_CFC_ (* Continuous Function Chart, elements in execution order *)
#0 RT_Pusk:R_TRIG(CLK: SCHU_P2_3_UST_RE_PUSK)
#1 TON_PCH_OTKL:TON(IN: SCHU_P2_3_UST_RE_STOP, PT: T#1s)
#2 FT_PCH_OTKL:R_TRIG(CLK: #1.Q)
#3 RS_YA1_Open:RS(SET: #0.Q, RESET1: #2.Q)
#4 ZADERJ_SHOD_YA1:TON(IN: #3.Q1, PT: t#10s)
#5 TON_YA1_Z_ZAM_TE2:TON(IN: SCHU_P2_3_TE2_M_ZASCH, PT: t#5s)
#6 OR(SCHU_P2_3_Z_M1_AV, NOT SCHU_P2_3_SA1_DI5_A)
#7 OR(SCHU_P2_3_Z_M2_AV, NOT SCHU_P2_3_SA8_DI3_A)
#8 AND(#6, #7)
#9 AND(NOT SCHU_P2_3_SA1_DI5_A, NOT SCHU_P2_3_SA8_DI3_A, NOT SCHU_P2_3_SA1_DI6_M, NOT SCHU_P2_3_SA8_DI4_M)
#10 OR(#8, #9)
#11 TON_OTK_MV:TON(IN: #10, PT: t#5s)
#12 OR(#5.Q, Z_ZAM_SR, #11.Q)
#13 SEL(SCHU_P2_3_SA7_DI1_A, eHVAC2PointActuatorMode_Close_OP, eHVAC2PointActuatorMode_Auto_BMS)
#14 SEL(#12, #13, eHVAC2PointActuatorMode_Close_OP)
#15 fb_HVACPA:FB_HVAC2PointActuator(eHVACDataSecurityType_Idle, FALSE, TRUE, #4.Q, #14, SCHU_P2_3_KV1_DI4, SCHU_P2_3_YA1_DI6_ZKR, SCHU_P2_3_YA1_DI7_OTK, TRUE, SCHU_P2_3_SB, enableLimitSwitch, stokeTime)
#16 SCHU_P2_3_SA7_DO7_OTK <= #15.out 1
#17 OR(#15.out 4, #15.out 5)
#18 YA1_OTKAZ <= #17
#19 INT_TO_TIME(SCHU_P2_3_YA1_VREMYA_HODA)
#20 MUL(#19, 1000)
#21 stokeTime <= #20
_END_CFC_
END_PROGRAM

(* POU IM/YA2_Upr, CFC *)
PROGRAM YA2_Upr
VAR
	YA2_PID: FB_HVACPIDCtrl;

	deadRange: REAL := 0.1;
	direction: BOOL;
	tTi: TIME;
	tTv: TIME;
	tTd: TIME;

	rYMin: REAL := 0;
	rYMax: REAL := 100;
	TON_SCHU_P2_3_P1_DI4_RUN: TON;
	reg1: BOOL;
	reg2: BOOL;

	SCHU_P2_3_YA2_: BOOL;
	YA2_REG_POL: BOOL;
	rwx: REAL;
	EPS1: REAL;
	EPS2: REAL;
END_VAR
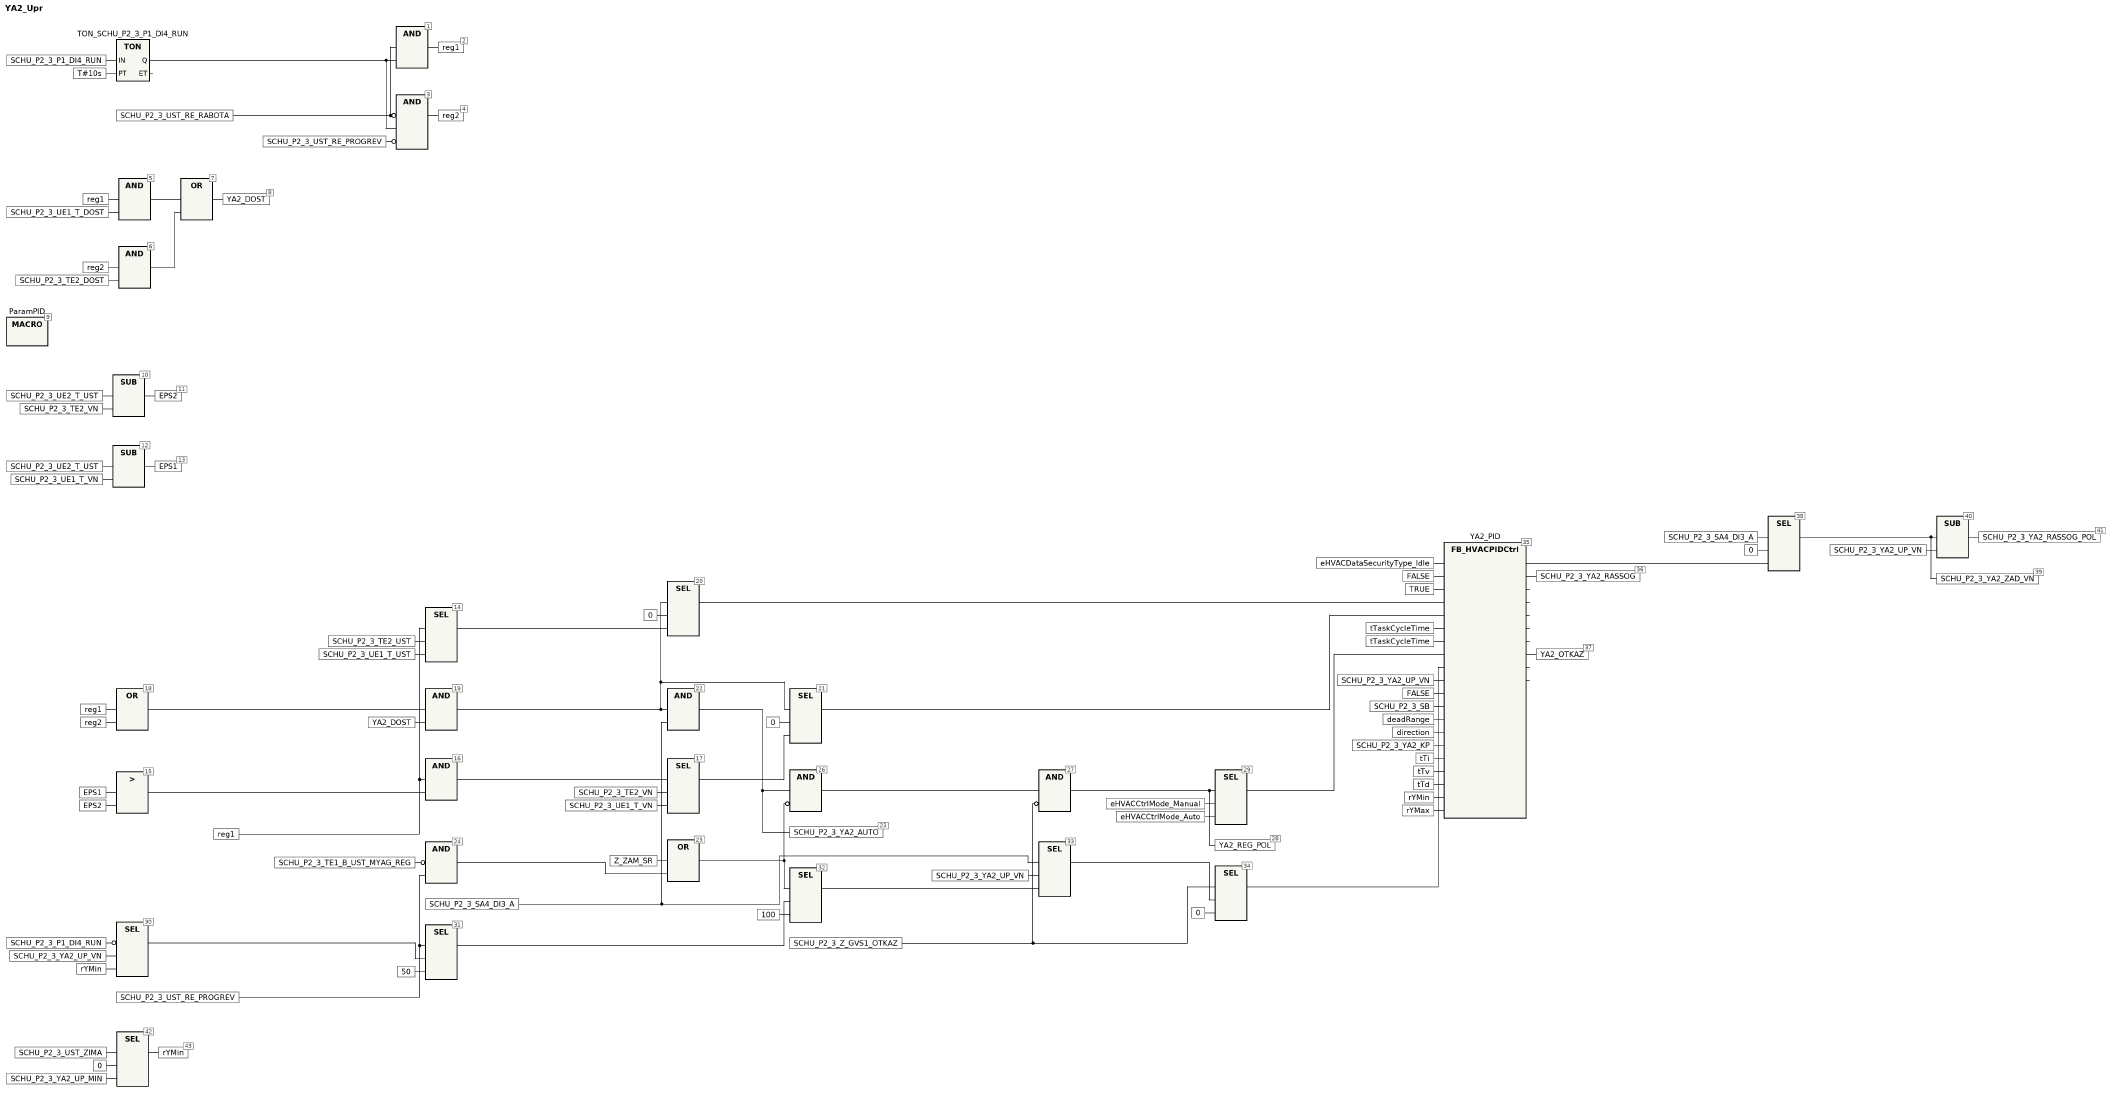
